// TIA Portal V20 export
// export: Created 2026-04-11T06:02:29.5928273Z, ExportSetting WithDefaults, DisplayName Totally Integrated Automation Portal, DisplayVersion V20, DisplayName TIA Portal Openness, DisplayVersion V20, DisplayName TIA Portal Version Control Interface, DisplayVersion V20, DisplayName STEP 7 Professional, DisplayVersion V20, DisplayName STEP 7 Safety, DisplayVersion V20, DisplayName WinCC Basic/Comfort/Advanced, DisplayVersion V20, DisplayName WinCC Unified, DisplayVersion V20
TYPE "udtHMI_SystemControl"
// stored: IsFailsafeCompliant false
   STRUCT
      iMode { S7_SetPoint := 'True'} : Int;   // System mode
      bEStop { ExternalWritable := 'False'} : Bool;   // System hardware E-Stop
      bError { ExternalWritable := 'False'} : Bool;   // Actuators error present
      bWarning { ExternalWritable := 'False'} : Bool;   // Warning present
      bAuto { ExternalWritable := 'False'} : Bool;   // All actuators in auto mode
      bPB_ResetError : Bool;   // Reset error push button
   END_STRUCT;
END_TYPE
